// TwinCAT 3 PLC project Test
// ProgramVersion: 3.1.4024.0
// libraries:
//   Tc2_Standard, * (Beckhoff Automation GmbH)
//   Tc2_System, * (Beckhoff Automation GmbH)
//   Tc3_Module, * (Beckhoff Automation GmbH)
// project tree:
//   / PlcTask.TcTTO
//   POUs/ MAIN.TcPOU

CONFIGURATION Test
    RESOURCE PLC ON TwinCAT3
        TASK PlcTask(INTERVAL := T#10ms, PRIORITY := 20);
        PROGRAM MAIN WITH PlcTask : MAIN;
    END_RESOURCE
END_CONFIGURATION

// ---- POUs/MAIN.TcPOU
PROGRAM MAIN
// Program başlangıç
VAR
    ButtonState : BOOL; // Buton durumu
    LampState : BOOL; // Lamba durumu
END_VAR

// Ana döngü

// Ana döngü
WHILE TRUE DO
    // Buton durumunu kontrol et
    ButtonState := ReadButtonState();

    // Buton basıldıysa
    IF ButtonState THEN
        // Lambayı aç
        LampState := TRUE;
    ELSE
        // Lambayı kapat
        LampState := FALSE;
    END_IF

END_PROGRAM
